PROGRAM P01_TwoPhasesBarriers
VAR_INPUT
IbBarrierBetweenWeightOpenedSensor 			AT %I*: BOOL;	
IbBarrierBetweenWeightClosedSensor 			AT %I*: BOOL;
IbBarrierBetweenDispencerOpenedSensor 		AT %I*: BOOL;
IbBarrierBetweenDispencerClosedSensor 		AT %I*: BOOL;
IbGateBeforeWeights56				 		AT %I*: BOOL;
END_VAR



VAR
	
	QbBarrierBetweenDispencerActuator 			: BOOL; 				 // Wyjście sterujące szlabanem ruchomym pod dozownikami
	//IbBarrierBetweenDispencerOpenedSensor 		AT %I*: BOOL; 			 // Wejście czujnika siłownika środkowej ruchomej bandy pod dozownikami
	//IbBarrierBetweenDispencerClosedSensor 		AT %I*: BOOL; 			 // Wejście czujnika siłownika środkowej ruchomej bandy pod dozownikami

	QbBarrierBetweenWeightActuator 			: BOOL; 				 // Wyjście sterujące szlabanem przed wagami
	
	//IbBarrierBetweenWeightOpenedSensor 			AT %I*: BOOL; 			// Wejście czujnika siłownika środkowej ruchomej bandy przed wjazdem na wagę
	//IbBarrierBetweenWeightClosedSensor 			AT %I*: BOOL; 			// Wejście czujnika siłownika środkowej ruchomej bandy przed wjazdem na wagę

	
	fbBarrierDispencer							: FB_Gate;				// Bloczek obsługi bandy 
	fbBarrierWeight								: FB_Gate;				// Bloczek obsługi bandy 	
	
	bTemp: BOOL;
END_VAR

aBeforeWeight();
aBetweenDispencer();

ACTION aBeforeWeight:
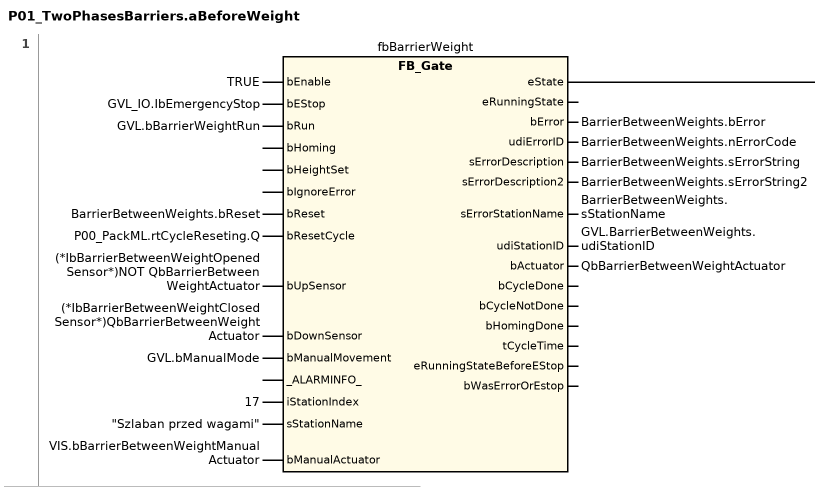
// NETWORK 1
fbBarrierWeight(
    bEnable := TRUE,
    bEStop := GVL_IO.IbEmergencyStop,
    bRun := GVL.bBarrierWeightRun,
    bReset := BarrierBetweenWeights.bReset,
    bResetCycle := P00_PackML.rtCycleReseting.Q,
    bUpSensor := (*IbBarrierBetweenWeightOpenedSensor*)NOT QbBarrierBetweenWeightActuator,
    bDownSensor := (*IbBarrierBetweenWeightClosedSensor*)QbBarrierBetweenWeightActuator,
    bManualMovement := GVL.bManualMode,
    iStationIndex := 17,
    sStationName := "Szlaban przed wagami",
    bManualActuator := VIS.bBarrierBetweenWeightManualActuator,
    bError => BarrierBetweenWeights.bError,
    udiErrorID => BarrierBetweenWeights.nErrorCode,
    sErrorDescription => BarrierBetweenWeights.sErrorString,
    sErrorDescription2 => BarrierBetweenWeights.sErrorString2,
    sErrorStationName => BarrierBetweenWeights.sStationName,
    udiStationID => GVL.BarrierBetweenWeights.udiStationID,
    bActuator => QbBarrierBetweenWeightActuator); // FB_Gate
END_ACTION

ACTION aBetweenDispencer:
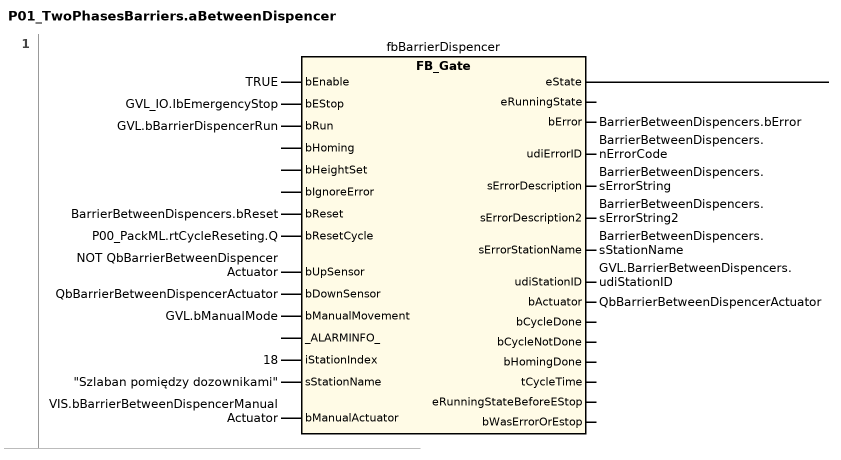
// NETWORK 1
fbBarrierDispencer(
    bEnable := TRUE,
    bEStop := GVL_IO.IbEmergencyStop,
    bRun := GVL.bBarrierDispencerRun,
    bReset := BarrierBetweenDispencers.bReset,
    bResetCycle := P00_PackML.rtCycleReseting.Q,
    bUpSensor := NOT QbBarrierBetweenDispencerActuator,
    bDownSensor := QbBarrierBetweenDispencerActuator,
    bManualMovement := GVL.bManualMode,
    iStationIndex := 18,
    sStationName := "Szlaban pomiędzy dozownikami",
    bManualActuator := VIS.bBarrierBetweenDispencerManualActuator,
    bError => BarrierBetweenDispencers.bError,
    udiErrorID => BarrierBetweenDispencers.nErrorCode,
    sErrorDescription => BarrierBetweenDispencers.sErrorString,
    sErrorDescription2 => BarrierBetweenDispencers.sErrorString2,
    sErrorStationName => BarrierBetweenDispencers.sStationName,
    udiStationID => GVL.BarrierBetweenDispencers.udiStationID,
    bActuator => QbBarrierBetweenDispencerActuator); // FB_Gate
END_ACTION

END_PROGRAM

(* stored: Version 1.1.0.1, ProductVersion 3.1.4026.13, FileIdentifier 7b08a60013dc5358c997c7a099b559343464c144, FileSignature 8f89b2a45e5fd6e7620cff9fb025811380567caf32a86767321d1db7e2ad4b0c2d95b3ae8ce814fd8b2dbbcd1b4a42ee1a067cf18a37634297e2e68a1c51da25f9ed6a2899946b3720f3241eeb266874d04ba62463bfc9ec1282088c6abdd1326fd6587261b48b57e4c4d56a0b46b3d028a9629643a3054e1dbf238d593f6ce932d50bfca9cf0ed1e7577d1f7e1efd4702ab7e6199dbd60baec122bccb8cb375f47eb3cea67fc3786a2c935223360c639ab484ffd6deef09d25b8f227e0569fcd9273f7876a3a527499b8798fb58e4970610d05e6dc452b0b5ad1cb13ba5b3d705b88f4216d0217cf63bdb3e2e9b763816dbba411324b81826bcd93b9792adee
   POU P01_TwoPhasesBarriers: Id {63126081-d1b4-4f1d-b274-bd71e640bd30}, SpecialFunc None
   Action aBeforeWeight: Id {d206367f-7d2c-4b7c-8111-c979be5d53e5}
   Action aBetweenDispencer: Id {0baf445b-6031-4640-9f92-a243e2917f1c} *)
